PROGRAM Calender
VAR
	DayNight: SR;
	calenderTimer: TON;
	AnotherOne: TON;
	Cycle: BOOL;
	Start: BOOL;
	On: BOOL;
	Morning: BOOL;
	HalfADay: TIME := T#25ms;
END_VAR

calenderTimer(IN:=Start , PT:= HalfADay, Q=> Cycle , ET=> );

IF Cycle = TRUE THEN
	GVL.Day := GVL.Day + 1;
	GVL.Cycle := TRUE;
	Start := FALSE;
ELSE
	GVL.Cycle := FALSE;
END_IF

AnotherOne(IN:=on AND NOT Start , PT:=HalfADay , Q=>Morning , ET=> );

DayNight(SET1:=Morning , RESET:=Cycle , Q1=>Start );

END_PROGRAM

(* stored: Version 1.1.0.1, ProductVersion 3.1.4024.12
   POU Calender: Id {481eedc4-1d9e-4340-907d-d6fb7a0ecc14}, SpecialFunc None *)
